// Mitsubishi GX Works2 project: SEQUENCE_REPEAT2   PLC: Q03UDV

PROGRAM MAIN
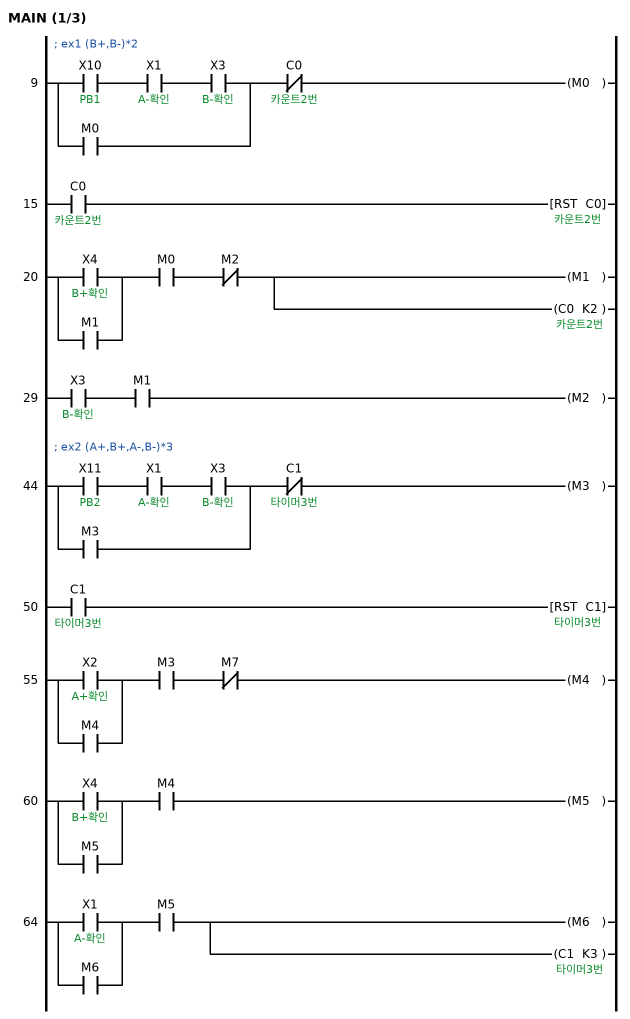
; ex1 (B+,B-)*2
9     LD      X10  ; PB1
      AND     X1  ; A-확인
      AND     X3  ; B-확인
      OR      M0
      ANI     C0  ; 카운트2번
      OUT     M0
15    LD      C0  ; 카운트2번
      RST     C0  ; 카운트2번
20    LD      X4  ; B+확인
      OR      M1
      AND     M0
      ANI     M2
      OUT     M1
      OUT     C0 K2  ; 카운트2번
29    LD      X3  ; B-확인
      AND     M1
      OUT     M2
; ex2 (A+,B+,A-,B-)*3
44    LD      X11  ; PB2
      AND     X1  ; A-확인
      AND     X3  ; B-확인
      OR      M3
      ANI     C1  ; 타이머3번
      OUT     M3
50    LD      C1  ; 타이머3번
      RST     C1  ; 타이머3번
55    LD      X2  ; A+확인
      OR      M4
      AND     M3
      ANI     M7
      OUT     M4
60    LD      X4  ; B+확인
      OR      M5
      AND     M4
      OUT     M5
64    LD      X1  ; A-확인
      OR      M6
      AND     M5
      OUT     M6
      OUT     C1 K3  ; 타이머3번
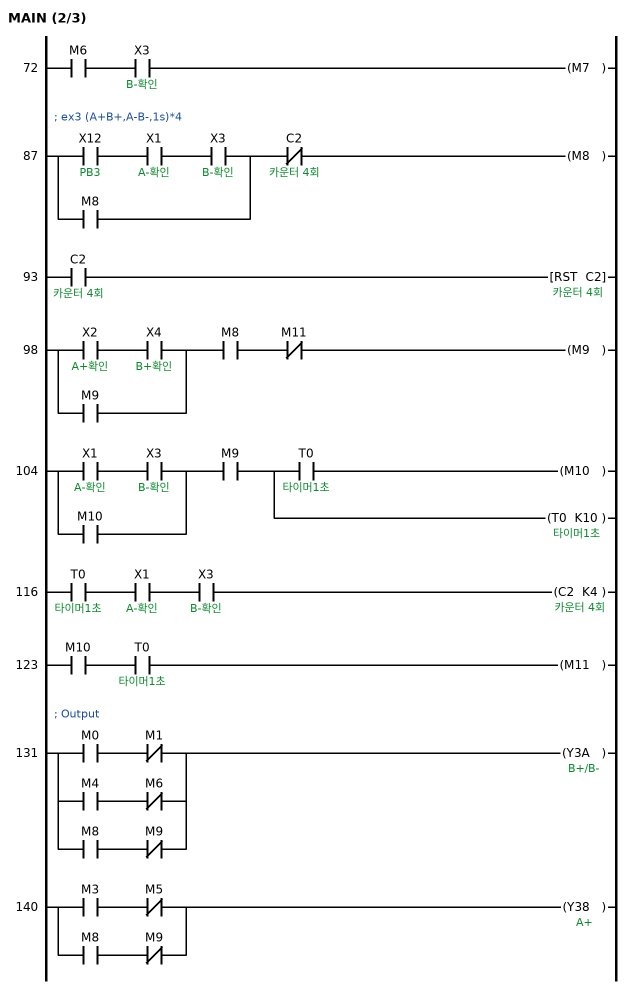
72    LD      M6
      AND     X3  ; B-확인
      OUT     M7
; ex3 (A+B+,A-B-,1s)*4
87    LD      X12  ; PB3
      AND     X1  ; A-확인
      AND     X3  ; B-확인
      OR      M8
      ANI     C2  ; 카운터 4회
      OUT     M8
93    LD      C2  ; 카운터 4회
      RST     C2  ; 카운터 4회
98    LD      X2  ; A+확인
      AND     X4  ; B+확인
      OR      M9
      AND     M8
      ANI     M11
      OUT     M9
104   LD      X1  ; A-확인
      AND     X3  ; B-확인
      OR      M10
      AND     M9
      MPS
      AND     T0  ; 타이머1초
      OUT     M10
      MPP
      OUT     T0 K10  ; 타이머1초
116   LD      T0  ; 타이머1초
      AND     X1  ; A-확인
      AND     X3  ; B-확인
      OUT     C2 K4  ; 카운터 4회
123   LD      M10
      AND     T0  ; 타이머1초
      OUT     M11
; Output
131   LD      M0
      ANI     M1
      LD      M4
      ANI     M6
      ORB
      LD      M8
      ANI     M9
      ORB
      OUT     Y3A  ; B+/B-
140   LD      M3
      ANI     M5
      LD      M8
      ANI     M9
      ORB
      OUT     Y38  ; A+
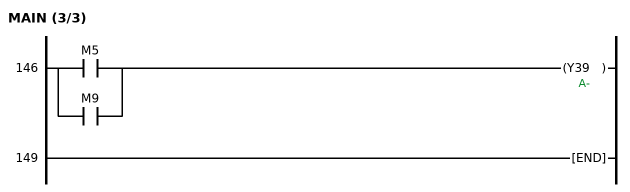
146   LD      M5
      OR      M9
      OUT     Y39  ; A-
149   END
END_PROGRAM
